PROGRAM F26_EncodersCtrl
VAR
	fbSingleTurnEncoder: FB_ENCODER_SingleTurn;
	fbTransferEncoder	: FB_ENCODER_AbsValueToPos;
	bStart: BOOL;
	nOutputRevolutions: UDINT := 0;
	nOutputPulses: UDINT;
	fOutputMM: REAL;

	nDummyEncoderPosition	: UDINT;
	nAlarmStatus		: UINT;
	nWarningStatus		: UINT;
END_VAR

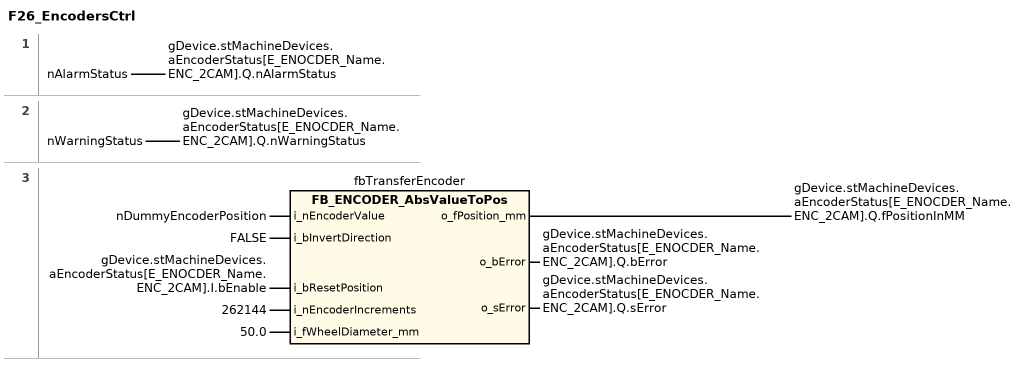
// NETWORK 1
gDevice.stMachineDevices.aEncoderStatus[E_ENOCDER_Name.ENC_2CAM].Q.nAlarmStatus := nAlarmStatus;

// NETWORK 2
gDevice.stMachineDevices.aEncoderStatus[E_ENOCDER_Name.ENC_2CAM].Q.nWarningStatus := nWarningStatus;

// NETWORK 3
fbTransferEncoder(
    i_nEncoderValue := nDummyEncoderPosition,
    i_bInvertDirection := FALSE,
    i_bResetPosition := gDevice.stMachineDevices.aEncoderStatus[E_ENOCDER_Name.ENC_2CAM].I.bEnable,
    i_nEncoderIncrements := 262144,
    i_fWheelDiameter_mm := 50.0,
    o_bError => gDevice.stMachineDevices.aEncoderStatus[E_ENOCDER_Name.ENC_2CAM].Q.bError,
    o_sError => gDevice.stMachineDevices.aEncoderStatus[E_ENOCDER_Name.ENC_2CAM].Q.sError); // FB_ENCODER_AbsValueToPos
gDevice.stMachineDevices.aEncoderStatus[E_ENOCDER_Name.ENC_2CAM].Q.fPositionInMM := fbTransferEncoder.o_fPosition_mm;

END_PROGRAM

(* stored: Version 1.1.0.1
   POU F26_EncodersCtrl: Id {47c32b3a-dc36-4c9f-95c3-40ea18c52ab2}, SpecialFunc None *)
